{attribute 'GeneratedUsingTerminal: EL4712--0000'}
{attribute addProperty BoxType "EL4712--0000"}
{attribute addProperty Id "Ch1_CycleCountAT %Q*UINT2"}
{attribute addProperty CRC "150317039"}
{attribute addProperty Size "2"}
TYPE Ch1_CycleCount_08F5A7EF :
STRUCT
	{attribute addProperty Name "Ch1_CycleCount"}
	Ch1_CycleCount AT %Q* : UINT;
END_STRUCT
END_TYPE

(* stored: Version 1.2.0.0, ProductVersion 3.1.4024.9
   DUT Ch1_CycleCount_08F5A7EF: Id {dcf4e1e3-2aa5-4d5c-8dfa-aaba3a896914} *)
